FUNCTION_BLOCK FB_StopMotion
VAR_INPUT
	bExecute      : BOOL := FALSE;
	rDeceleration : LREAL;
END_VAR
VAR_IN_OUT
	Axis         : AXIS_REF;
END_VAR
VAR_OUTPUT
	bStopDone	: BOOL := FALSE;
	bStopError	: BOOL := FALSE;
	bStopBusy	: BOOL := FALSE;
END_VAR
VAR
	fbStop	: MC_Stop;
END_VAR

fbStop(
	Axis         := Axis,
	Execute      := bExecute,  
	Deceleration := 10.0,
	Busy 		 => bStopBusy
);
IF fbStop.Done AND NOT fbStop.Error THEN
	bStopDone 	:= TRUE;
	bStopError	:= FALSE;
END_IF
IF fbStop.Error THEN
	bStopDone 	:= FALSE;
	bStopError	:= TRUE;
END_IF

END_FUNCTION_BLOCK

(* stored: Version 1.1.0.1, ProductVersion 3.1.4024.12
   POU FB_StopMotion: Id {6250a62b-82b3-4c7f-b0dc-6739d5bed503}, SpecialFunc None *)
